FUNCTION_BLOCK PUBLIC FB_CDPlayer
VAR_OUTPUT
	bPlayerActive		: BOOL;
	byVolume			: BYTE;
	byTrack				: UINT;
END_VAR

PROPERTY PUBLIC PlayerActive : BOOL
GET
PlayerActive := bPlayerActive;
END_GET
END_PROPERTY

METHOD PUBLIC SetTrack : BOOL
VAR_INPUT
	byNewTrack			:	UINT;
END_VAR
byTrack := byNewTrack;
END_METHOD

METHOD PUBLIC SetVolume : BOOL
VAR_INPUT
	byNewVolume 		: BYTE;
END_VAR
byVolume := byNewVolume;
END_METHOD

METHOD PUBLIC Start
bPlayerActive := true;
END_METHOD

METHOD PUBLIC Stop
bPlayerActive := FALSE;
END_METHOD

PROPERTY PUBLIC Track : UINT
GET
Track := byTrack;
END_GET
END_PROPERTY

PROPERTY PUBLIC Volume : BYTE
GET
Volume := byVolume;
END_GET
END_PROPERTY

END_FUNCTION_BLOCK

(* stored: Version 1.1.0.1, ProductVersion 3.1.4024.12
   POU FB_CDPlayer: Id {053e9744-dade-46b5-bd05-c0670f467c64}, SpecialFunc None
   Property PlayerActive: Id {39846a2b-1c17-4a3c-94a2-d01421974622}
   Get Get: Id {0a82b6f3-0650-4b76-9bd0-de68689ec643}
   Method SetTrack: Id {37acc586-6784-4cea-b82a-0e0ae11fbbaf}
   Method SetVolume: Id {c7139fca-157c-4fdb-a12a-0b9eb2889f17}
   Method Start: Id {3d4a8917-9407-4a29-970b-7c9ebed329ff}
   Method Stop: Id {b92fa661-c5af-4cc4-8932-478a96b318b6}
   Property Track: Id {5abf2943-f6a5-44c8-a98c-b8474b3d7da7}
   Get Get: Id {1f96d752-8bec-4461-801e-8864956ee484}
   Property Volume: Id {254cf412-4c21-4b9b-a0ae-020e68afac1c}
   Get Get: Id {99c4f109-cbd9-4639-b04e-4e52f380cfff} *)
